FUNCTION_BLOCK ABSTRACT FB_ActorContinous EXTENDS FB_Actor2Point
VAR_INPUT
	//internal input variables:
	fSetPointAutomatic	: REAL; //set setpoint in percent 0.0 - 100.0
END_VAR
VAR_OUTPUT
END_VAR
VAR
	//OPC UA structured variables:
	{attribute 'OPC.UA.DA' := '1'}
	setSetPoint : ST_SetSetPoint;
	{attribute 'OPC.UA.DA' := '1'}
	setPointState : ST_SetPointState;
	
	//internal variables:
	fSetPoint : REAL; //actual set setpoint in percent 0.0 - 100.0
	aSetPointLimits	: ARRAY[1..2] OF REAL := [0, 100]; //lower and upper set point limit
END_VAR

PROPERTY fLowerSetPointLimit : REAL; //set lower set point limit
GET
fLowerSetPointLimit := aSetPointLimits[1];
END_GET
SET
aSetPointLimits[1] := fLowerSetPointLimit;
setPointState.aSetPointLimits := aSetPointLimits;
END_SET
END_PROPERTY

PROPERTY fUpperSetPointLimit : REAL //set upper set point limit
GET
fUpperSetPointLimit := aSetPointLimits[2];
END_GET
SET
aSetPointLimits[2] := fUpperSetPointLimit;
setPointState.aSetPointLimits := aSetPointLimits;
END_SET
END_PROPERTY

METHOD PROTECTED MAIN : BOOL // Method that calls all needed function block methods
VAR_INPUT
END_VAR
SelectControlMode();
SelectSetPoint();
SetPointCheck();
END_METHOD

METHOD PROTECTED FINAL SelectControlMode : BOOL
VAR_INPUT
END_VAR
SUPER^.SelectControlMode();

//add changing set point to method
IF control.bManualModeActivated THEN
	fsetPoint := setSetPoint.fSetPointManual;
ELSIF control.bAlgorithmModeActivated AND algorithmPermission THEN
	fsetPoint := setSetPoint.fSetPointAlgorithm;
ELSE
	fsetPoint := fSetPointAutomatic;
END_IF
END_METHOD

METHOD PROTECTED FINAL SelectSetPoint : BOOL
VAR_INPUT
END_VAR
//change access mode
IF control.bManualModeActivated THEN
	fsetPoint := setSetPoint.fSetPointManual;
ELSIF control.bAlgorithmModeActivated AND algorithmPermission THEN
	fsetPoint := setSetPoint.fSetPointAlgorithm;
ELSE
	fsetPoint := fSetPointAutomatic;
END_IF
setPointState.fSetPoint := fSetPoint;
END_METHOD

METHOD PROTECTED FINAL SetPointCheck : BOOL
VAR
	aLocalSetPointLimits : ARRAY[1..2] OF REAL := aSetPointLimits;
END_VAR
//control value must not be below the lower limit
fSetPoint := MAX(fSetPoint, aLocalSetPointLimits[1]);

//control value must not be above the upper limit
fSetPoint := MIN(fSetPoint, aLocalSetPointLimits[2]);
END_METHOD

END_FUNCTION_BLOCK

(* stored: Version 1.1.0.1, ProductVersion 3.1.4024.9
   POU FB_ActorContinous: Id {c8bff7e9-c02c-4471-8259-14c86f2cd564}, SpecialFunc None
   Property fLowerSetPointLimit: Id {796dd9fb-c52d-4acd-9fa6-dc7e631b498d}
   Get Get: Id {dfc88d31-f790-4b77-86cd-90806c52cfb4}
   Set Set: Id {eb1ec4b7-b0b3-49de-b291-c6ccce0d6210}
   Property fUpperSetPointLimit: Id {fb4707ce-856d-497a-a2f5-99887319386f}
   Get Get: Id {75fedf8f-b247-42bc-bba6-2e70fb22bf6e}
   Set Set: Id {a00ba8d7-fa9c-4009-8dbd-de57d102b8e3}
   Method MAIN: Id {7c71e98c-e88b-49de-b162-405ba243d74c}
   Method SelectControlMode: Id {9487b088-9bc5-4a7e-8bf7-9767eafe3f05}
   Method SelectSetPoint: Id {c00b1980-2db2-4070-bc69-4d3e586d5c0d}
   Method SetPointCheck: Id {a788f595-bc97-42ed-a5e1-110d1f06de83} *)
